// TIA Portal V16 export
// export: Created 2022-11-14T17:35:29.674924Z, ExportSetting WithDefaults, DisplayName Totally Integrated Automation Portal, DisplayVersion V16, DisplayName TIA Portal Version Control Interface, DisplayVersion V16, DisplayName TIA Portal Openness, DisplayVersion V16, DisplayName STEP 7 Professional, DisplayVersion V16, DisplayName STEP 7 Safety, DisplayVersion V16, DisplayName WinCC Advanced, DisplayVersion V16
FUNCTION "FC42_RopeUnit" : Void   // FC42, LAD
TITLE = RopeUnit
{ S7_Optimized_Access := 'FALSE' }
VERSION : 0.1
// stored: AutoNumber false, IsIECCheckEnabled false, SetENOAutomatically false, UDAEnableTagReadback false
   VAR_TEMP
      OpenCloseDoubleRope : Bool;
      DoubleRopeOpen : Bool;
      TempInt : Int;
      TempInt1 : Int;
   END_VAR
   VAR_TEMP   // added for the SCL form of the ladder/FBD networks
      _w1 : Bool;
   END_VAR
BEGIN

REGION Network 1: Timeout for single or lower(double) rope unit open/close
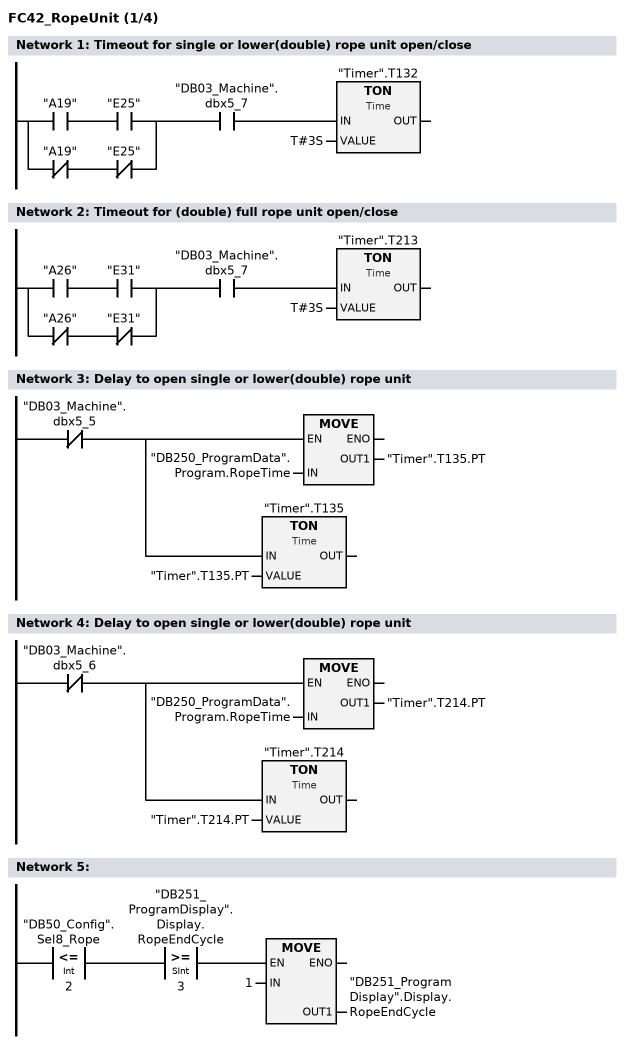
   "Timer".T132.TON(IN := (("A19" AND "E25") OR (NOT "A19" AND NOT "E25")) AND "DB03_Machine".dbx5_7, PT := T#3S);   // TON coil
END_REGION

REGION Network 2: Timeout for (double) full rope unit open/close
   "Timer".T213.TON(IN := (("A26" AND "E31") OR (NOT "A26" AND NOT "E31")) AND "DB03_Machine".dbx5_7, PT := T#3S);   // TON coil
END_REGION

REGION Network 3: Delay to open single or lower(double) rope unit
   #_w1 := NOT "DB03_Machine".dbx5_5;
   IF #_w1 THEN "Timer".T135.PT := "DB250_ProgramData".Program.RopeTime; END_IF;
   "Timer".T135.TON(IN := #_w1, PT := "Timer".T135.PT);   // TON coil
END_REGION

REGION Network 4: Delay to open single or lower(double) rope unit
   #_w1 := NOT "DB03_Machine".dbx5_6;
   IF #_w1 THEN "Timer".T214.PT := "DB250_ProgramData".Program.RopeTime; END_IF;
   "Timer".T214.TON(IN := #_w1, PT := "Timer".T214.PT);   // TON coil
END_REGION

REGION Network 5
   RUNG wire#powerrail
      { S7_Templates := "SrcType := Int" } LE_Contact(in1 := "DB50_Config".Sel8_Rope, in2 := 2)
      { S7_Templates := "SrcType := SInt" } GE_Contact(in1 := "DB251_ProgramDisplay".Display.RopeEndCycle, in2 := 3)
      { S7_GenerateENO := "TRUE" } Move(in := 1, out1 => "DB251_ProgramDisplay".Display.RopeEndCycle)
   END_RUNG
   // the same network as SCL:
   IF ("DB50_Config".Sel8_Rope <= 2) AND ("DB251_ProgramDisplay".Display.RopeEndCycle >= 3) THEN
       "DB251_ProgramDisplay".Display.RopeEndCycle := 1;
   END_IF;
END_REGION

REGION Network 6: RopeUnitOk1: Rope unit open
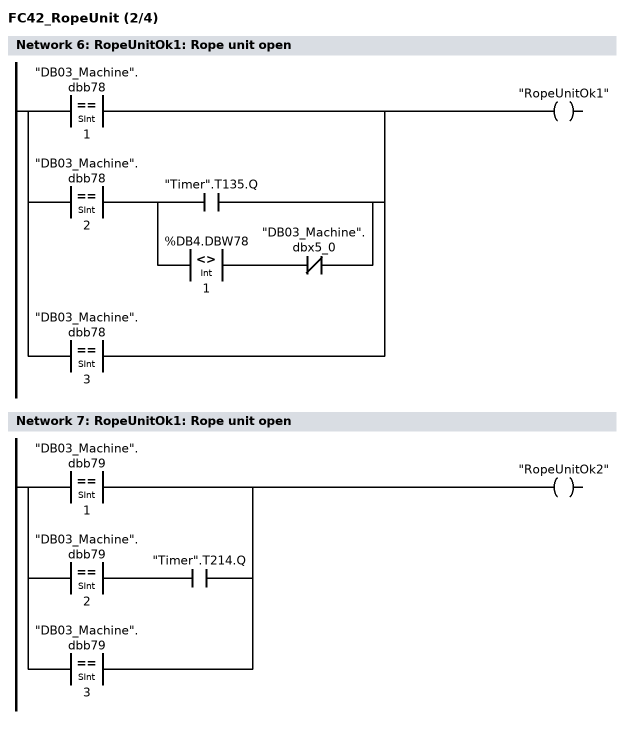
   RUNG wire#powerrail
      { S7_Templates := "SrcType := SInt" } EQ_Contact(in1 := "DB03_Machine".dbb78, in2 := 1)
      wire#w1
      Coil( "RopeUnitOk1" )
   END_RUNG
   RUNG wire#powerrail
      { S7_Templates := "SrcType := SInt" } EQ_Contact(in1 := "DB03_Machine".dbb78, in2 := 2)
      wire#w2
      Contact( "Timer".T135.Q )
   END_RUNG wire#w1
   RUNG wire#w2
      { S7_Templates := "SrcType := Int" } NE_Contact(in1 := %DB4.DBW78, in2 := 1)
      I_Contact( "DB03_Machine".dbx5_0 )
   END_RUNG wire#w1
   RUNG wire#powerrail
      { S7_Templates := "SrcType := SInt" } EQ_Contact(in1 := "DB03_Machine".dbb78, in2 := 3)
   END_RUNG wire#w1
   // the same network as SCL:
   "RopeUnitOk1" := ("DB03_Machine".dbb78 = 1) OR (("DB03_Machine".dbb78 = 2) AND ("Timer".T135.Q OR ((%DB4.DBW78 <> 1) AND NOT "DB03_Machine".dbx5_0))) OR ("DB03_Machine".dbb78 = 3);
END_REGION

REGION Network 7: RopeUnitOk1: Rope unit open
   RUNG wire#powerrail
      { S7_Templates := "SrcType := SInt" } EQ_Contact(in1 := "DB03_Machine".dbb79, in2 := 1)
      wire#w1
      Coil( "RopeUnitOk2" )
   END_RUNG
   RUNG wire#powerrail
      { S7_Templates := "SrcType := SInt" } EQ_Contact(in1 := "DB03_Machine".dbb79, in2 := 2)
      Contact( "Timer".T214.Q )
   END_RUNG wire#w1
   RUNG wire#powerrail
      { S7_Templates := "SrcType := SInt" } EQ_Contact(in1 := "DB03_Machine".dbb79, in2 := 3)
   END_RUNG wire#w1
   // the same network as SCL:
   "RopeUnitOk2" := ("DB03_Machine".dbb79 = 1) OR (("DB03_Machine".dbb79 = 2) AND "Timer".T214.Q) OR ("DB03_Machine".dbb79 = 3);
END_REGION

REGION Network 8: Closing upper(double) rope unit
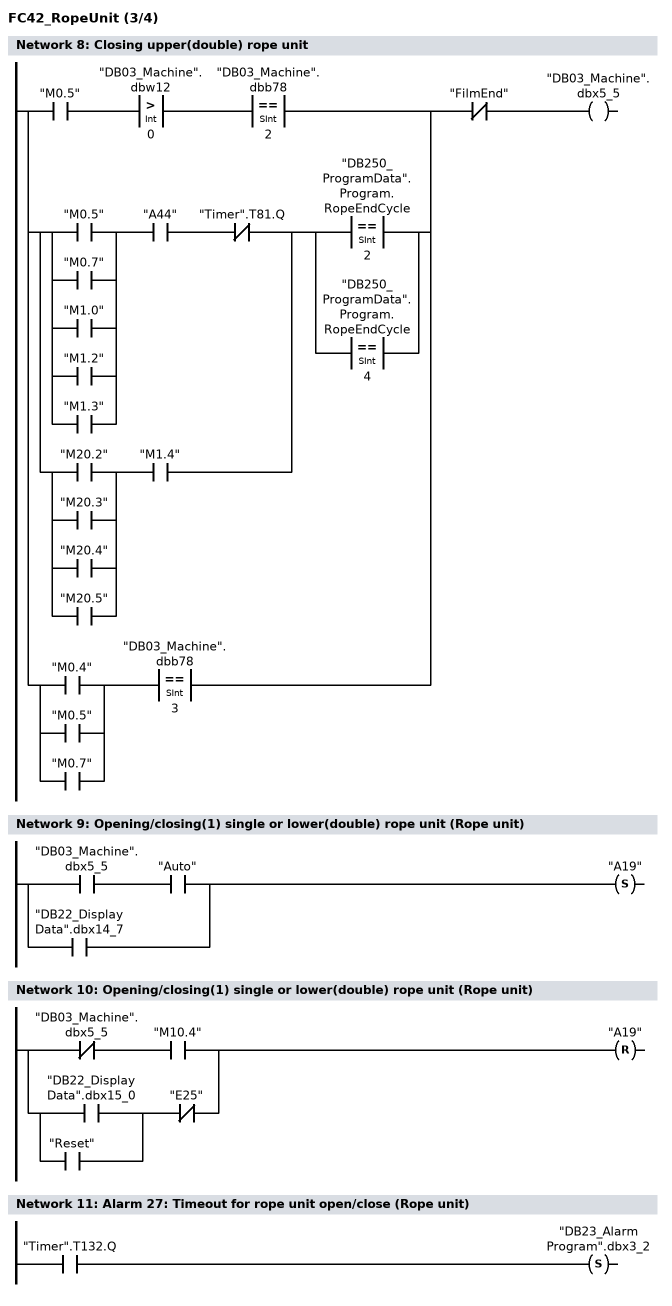
   RUNG wire#powerrail
      Contact( "M0.5" )
      { S7_Templates := "SrcType := Int" } GT_Contact(in1 := "DB03_Machine".dbw12, in2 := 0)
      { S7_Templates := "SrcType := SInt" } EQ_Contact(in1 := "DB03_Machine".dbb78, in2 := 2)
      wire#w1
      I_Contact( "FilmEnd" )
      Coil( "DB03_Machine".dbx5_5 )
   END_RUNG
   RUNG wire#powerrail
      Contact( "M0.5" )
      wire#w2
      Contact( "A44" )
      I_Contact( "Timer".T81.Q )
      wire#w3
      { S7_Templates := "SrcType := SInt" } EQ_Contact(in1 := "DB250_ProgramData".Program.RopeEndCycle, in2 := 2)
   END_RUNG wire#w1
   RUNG wire#powerrail
      Contact( "M0.7" )
   END_RUNG wire#w2
   RUNG wire#powerrail
      Contact( "M1.0" )
   END_RUNG wire#w2
   RUNG wire#powerrail
      Contact( "M1.2" )
   END_RUNG wire#w2
   RUNG wire#powerrail
      Contact( "M1.3" )
   END_RUNG wire#w2
   RUNG wire#powerrail
      Contact( "M20.2" )
      wire#w4
      Contact( "M1.4" )
   END_RUNG wire#w3
   RUNG wire#powerrail
      Contact( "M20.3" )
   END_RUNG wire#w4
   RUNG wire#powerrail
      Contact( "M20.4" )
   END_RUNG wire#w4
   RUNG wire#powerrail
      Contact( "M20.5" )
   END_RUNG wire#w4
   RUNG wire#w3
      { S7_Templates := "SrcType := SInt" } EQ_Contact(in1 := "DB250_ProgramData".Program.RopeEndCycle, in2 := 4)
   END_RUNG wire#w1
   RUNG wire#powerrail
      Contact( "M0.4" )
      wire#w5
      { S7_Templates := "SrcType := SInt" } EQ_Contact(in1 := "DB03_Machine".dbb78, in2 := 3)
   END_RUNG wire#w1
   RUNG wire#powerrail
      Contact( "M0.5" )
   END_RUNG wire#w5
   RUNG wire#powerrail
      Contact( "M0.7" )
   END_RUNG wire#w5
   // the same network as SCL:
   "DB03_Machine".dbx5_5 := (("M0.5" AND ("DB03_Machine".dbw12 > 0) AND ("DB03_Machine".dbb78 = 2)) OR (((("M0.5" OR "M0.7" OR "M1.0" OR "M1.2" OR "M1.3") AND "A44" AND NOT "Timer".T81.Q) OR (("M20.2" OR "M20.3" OR "M20.4" OR "M20.5") AND "M1.4")) AND (("DB250_ProgramData".Program.RopeEndCycle = 2) OR ("DB250_ProgramData".Program.RopeEndCycle = 4))) OR (("M0.4" OR "M0.5" OR "M0.7") AND ("DB03_Machine".dbb78 = 3))) AND NOT "FilmEnd";
END_REGION

REGION Network 9: Opening/closing(1) single or lower(double) rope unit (Rope unit)
   RUNG wire#powerrail
      Contact( "DB03_Machine".dbx5_5 )
      Contact( "Auto" )
      wire#w1
      S_Coil( "A19" )
   END_RUNG
   RUNG wire#powerrail
      Contact( "DB22_DisplayData".dbx14_7 )
   END_RUNG wire#w1
   // the same network as SCL:
   IF ("DB03_Machine".dbx5_5 AND "Auto") OR "DB22_DisplayData".dbx14_7 THEN "A19" := TRUE; END_IF;
END_REGION

REGION Network 10: Opening/closing(1) single or lower(double) rope unit (Rope unit)
   RUNG wire#powerrail
      I_Contact( "DB03_Machine".dbx5_5 )
      Contact( "M10.4" )
      wire#w1
      R_Coil( "A19" )
   END_RUNG
   RUNG wire#powerrail
      Contact( "DB22_DisplayData".dbx15_0 )
      wire#w2
      I_Contact( "E25" )
   END_RUNG wire#w1
   RUNG wire#powerrail
      Contact( "Reset" )
   END_RUNG wire#w2
   // the same network as SCL:
   IF (NOT "DB03_Machine".dbx5_5 AND "M10.4") OR (("DB22_DisplayData".dbx15_0 OR "Reset") AND NOT "E25") THEN
       "A19" := FALSE;
   END_IF;
END_REGION

REGION Network 11: Alarm 27: Timeout for rope unit open/close (Rope unit)
   RUNG wire#powerrail
      Contact( "Timer".T132.Q )
      S_Coil( "DB23_AlarmProgram".dbx3_2 )
   END_RUNG
   // the same network as SCL:
   IF "Timer".T132.Q THEN "DB23_AlarmProgram".dbx3_2 := TRUE; END_IF;
END_REGION

REGION Network 12: Closing upper(double) rope unit
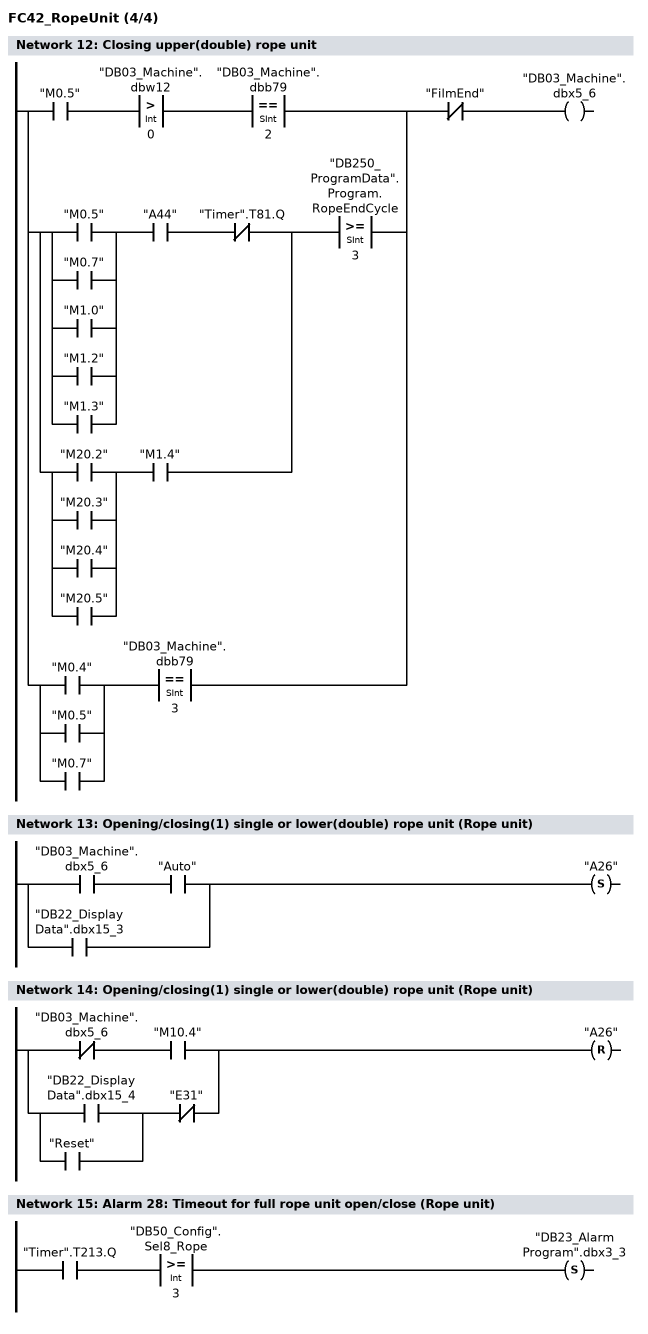
   RUNG wire#powerrail
      Contact( "M0.5" )
      { S7_Templates := "SrcType := Int" } GT_Contact(in1 := "DB03_Machine".dbw12, in2 := 0)
      { S7_Templates := "SrcType := SInt" } EQ_Contact(in1 := "DB03_Machine".dbb79, in2 := 2)
      wire#w1
      I_Contact( "FilmEnd" )
      Coil( "DB03_Machine".dbx5_6 )
   END_RUNG
   RUNG wire#powerrail
      Contact( "M0.5" )
      wire#w2
      Contact( "A44" )
      I_Contact( "Timer".T81.Q )
      wire#w3
      { S7_Templates := "SrcType := SInt" } GE_Contact(in1 := "DB250_ProgramData".Program.RopeEndCycle, in2 := 3)
   END_RUNG wire#w1
   RUNG wire#powerrail
      Contact( "M0.7" )
   END_RUNG wire#w2
   RUNG wire#powerrail
      Contact( "M1.0" )
   END_RUNG wire#w2
   RUNG wire#powerrail
      Contact( "M1.2" )
   END_RUNG wire#w2
   RUNG wire#powerrail
      Contact( "M1.3" )
   END_RUNG wire#w2
   RUNG wire#powerrail
      Contact( "M20.2" )
      wire#w4
      Contact( "M1.4" )
   END_RUNG wire#w3
   RUNG wire#powerrail
      Contact( "M20.3" )
   END_RUNG wire#w4
   RUNG wire#powerrail
      Contact( "M20.4" )
   END_RUNG wire#w4
   RUNG wire#powerrail
      Contact( "M20.5" )
   END_RUNG wire#w4
   RUNG wire#powerrail
      Contact( "M0.4" )
      wire#w5
      { S7_Templates := "SrcType := SInt" } EQ_Contact(in1 := "DB03_Machine".dbb79, in2 := 3)
   END_RUNG wire#w1
   RUNG wire#powerrail
      Contact( "M0.5" )
   END_RUNG wire#w5
   RUNG wire#powerrail
      Contact( "M0.7" )
   END_RUNG wire#w5
   // the same network as SCL:
   "DB03_Machine".dbx5_6 := (("M0.5" AND ("DB03_Machine".dbw12 > 0) AND ("DB03_Machine".dbb79 = 2)) OR (((("M0.5" OR "M0.7" OR "M1.0" OR "M1.2" OR "M1.3") AND "A44" AND NOT "Timer".T81.Q) OR (("M20.2" OR "M20.3" OR "M20.4" OR "M20.5") AND "M1.4")) AND ("DB250_ProgramData".Program.RopeEndCycle >= 3)) OR (("M0.4" OR "M0.5" OR "M0.7") AND ("DB03_Machine".dbb79 = 3))) AND NOT "FilmEnd";
END_REGION

REGION Network 13: Opening/closing(1) single or lower(double) rope unit (Rope unit)
   RUNG wire#powerrail
      Contact( "DB03_Machine".dbx5_6 )
      Contact( "Auto" )
      wire#w1
      S_Coil( "A26" )
   END_RUNG
   RUNG wire#powerrail
      Contact( "DB22_DisplayData".dbx15_3 )
   END_RUNG wire#w1
   // the same network as SCL:
   IF ("DB03_Machine".dbx5_6 AND "Auto") OR "DB22_DisplayData".dbx15_3 THEN "A26" := TRUE; END_IF;
END_REGION

REGION Network 14: Opening/closing(1) single or lower(double) rope unit (Rope unit)
   RUNG wire#powerrail
      I_Contact( "DB03_Machine".dbx5_6 )
      Contact( "M10.4" )
      wire#w1
      R_Coil( "A26" )
   END_RUNG
   RUNG wire#powerrail
      Contact( "DB22_DisplayData".dbx15_4 )
      wire#w2
      I_Contact( "E31" )
   END_RUNG wire#w1
   RUNG wire#powerrail
      Contact( "Reset" )
   END_RUNG wire#w2
   // the same network as SCL:
   IF (NOT "DB03_Machine".dbx5_6 AND "M10.4") OR (("DB22_DisplayData".dbx15_4 OR "Reset") AND NOT "E31") THEN
       "A26" := FALSE;
   END_IF;
END_REGION

REGION Network 15: Alarm 28: Timeout for full rope unit open/close (Rope unit)
   RUNG wire#powerrail
      Contact( "Timer".T213.Q )
      { S7_Templates := "SrcType := Int" } GE_Contact(in1 := "DB50_Config".Sel8_Rope, in2 := 3)
      S_Coil( "DB23_AlarmProgram".dbx3_3 )
   END_RUNG
   // the same network as SCL:
   IF "Timer".T213.Q AND ("DB50_Config".Sel8_Rope >= 3) THEN "DB23_AlarmProgram".dbx3_3 := TRUE; END_IF;
END_REGION
END_FUNCTION
